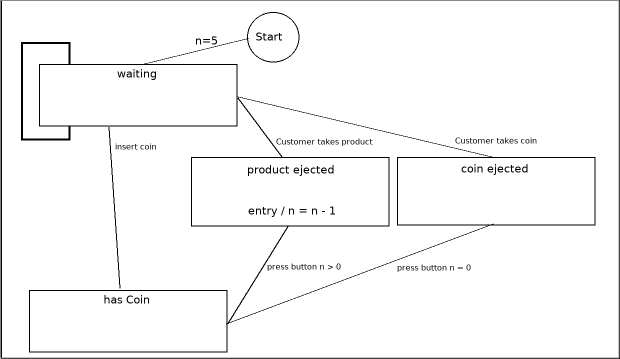
VISUALIZATION stateDiagramm  // 620x359
VAR_IN_OUT
	Panel		: POINTER TO ST_Panel;
END_VAR
    Rectangle (14,55 52x80)
    Rectangle (1,0 619x359)
    Ellipse (247,12 52x50)
    RoundedRectangle (29,290 198x62), colour toggle: Panel^.State='HasCoin'
    RoundedRectangle (191,157 198x69), colour toggle: Panel^.State='ProductEjected'
    RoundedRectangle (397,157 198x68), colour toggle: Panel^.State='CoinEjected'
    Line (228,323) (288,226)
    Line (493,224) (226,324)
    Line (282,157) (238,98)
    Line (236,96) (494,157)
    Line (120,288) (109,127)
    Label (32,285 190x30), "has Coin"
    Label (196,155 190x30), "product ejected"
    Label (400,154 190x30), "coin ejected"
    Label (197,196 190x30), "entry / n = n - 1"
    Line (134,66) (248,38)
    Label (245,22 48x30), "Start"
    Label (186,26 41x30), "n=5"
    Label (95,132 82x30), "insert coin"
    Rectangle (21,42 49x98)
    RoundedRectangle (39,64 198x62), colour toggle: (Panel^.State='Waiting')
    Label (62,59 150x30), "waiting"
    Label (391,253 86x30), "press button n = 0"
    Label (264,252 80x30), "press button n > 0"
    Label (272,127 105x30), "Customer takes product"
    Label (448,126 96x30), "Customer takes coin"
END_VISUALIZATION

(* stored: Version 1.1.0.1, ProductVersion 3.1.4024.9
   Visu stateDiagramm: Id {081c6ae1-f335-4321-8fec-4625bf1a7acd} *)
